# EPICS autosave request: ez4axis_example/as/req/all_motor_positions.req
file "motor_positions.req", P=$(P), M=m1
file "motor_positions.req", P=$(P), M=m2
file "motor_positions.req", P=$(P), M=m3
file "motor_positions.req", P=$(P), M=m4
